(* PLC project Unnamed, Неизвестно Unnamed 1 *)
(* stored: creationDateTime 2024-04-13T14:02:33, modificationDateTime 2024-04-13T14:08:33 *)

PROGRAM OLIA_test
  VAR
    TestVar AT %QW0 : DINT := 0;
  END_VAR
  VAR  (* added by the conversion: wires and edge detectors of the diagram *)
    _ADD2_OUT : DINT;
  END_VAR

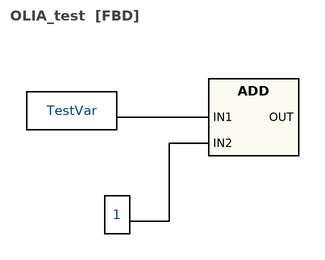
(* FBD diagram, written out as Structured Text *)
_ADD2_OUT := TestVar + 1;
END_PROGRAM

CONFIGURATION Config0
  RESOURCE Res0 ON PLC
    TASK task0(INTERVAL := T#20ms, PRIORITY := 0);
    PROGRAM instance0 WITH task0 : OLIA_test;
  END_RESOURCE
END_CONFIGURATION
